Fanuc KAREL source: kt00923.KL

-- PROVISIONAL review KL for V940-1; original PC SHA256 790fc730eb016748a5e325f3f7eaf1c4d983b5ac3d3b56decbed80735e3515d1
-- Incomplete behavior may be omitted. Consult companion uncertainty JSON. Do not deploy.
PROGRAM KT00923
%NOLOCKGROUP
VAR
  S1 : STRING[80]
  S2 : STRING[80]
  OUT : STRING[80]
BEGIN
  -- V9_ZERO_TABLE_METADATA_HINT layout=0001; no indexed target words; source/name/runtime held
  -- UNRESOLVED_PC offsets 5-14; opcodes 3F,75
  -- UNRESOLVED_PC offsets 19-28; opcodes 3F,75
  -- UNRESOLVED_PC offsets 33-42; opcodes 3F,75
  -- UNRESOLVED_PC offsets 47-56; opcodes 3F,75
  -- UNRESOLVED_PC offsets 61-82; opcodes 27,22,2A,27,9D,27,9D,76,75
  -- UNRESOLVED_PC offsets 87-91; opcodes 7F
END KT00923
